(* Logix 5000 project; controller WWTP_SOLIDS_CLX vendor 1 type 14 code 54 rev 17.2; software revision 17.00; part 13 of 16 *)
(* tags used below, declared in another part *)
   Inp_ActuatorFault : BOOL;   // Valve Actuator Fault (overload, etc.), 0=OK, 1=Fault)
   Inp_OpenPermOK : BOOL;   // 1=Open Permissives OK, Valve can motor open
   Inp_OpenNBPermOK : BOOL;   // 1=Non-Bypassable Open Permissives OK, valve can motor open
   Inp_ClosePermOK : BOOL;   // 1=Close Permissives OK, Valve can motor closed
   Inp_CloseNBPermOK : BOOL;   // 1=Non-Bypassable Close Permissives OK, valve can motor closed
   Inp_IOFault : BOOL;   // Input Communication Status 0=OK, 1=fail
   Inp_Sim : BOOL;   // 1=Simulate working valve; 0=Open/Close/ Monitor actual valve
   Cfg_UseOpenLS : BOOL;   // 1=Valve Open LS should be used for failure checking
   Cfg_UseClosedLS : BOOL;   // 1=Valve Closed LS should be used for failure checking
   Cfg_HasStop : BOOL;   // 1=Stop output can be used to break local seal-in and stop valve motion
   Cfg_PCmdClear : BOOL;   // 1=Clear Program Commands on receipt 0=Leave Set
   Cfg_HasFullStallAlm : BOOL;   // 1=Full Stall Alarm exists and will be checked
   Cfg_HasTransitStallAlm : BOOL;   // 1=Transit Stall Alarm exists and will be checked
   Cfg_HasActuatorFaultAlm : BOOL;   // 1=Actuator Fault Alarm exists and will be checked
   Cfg_HasIOFaultAlm : BOOL;   // 1=I/O Fault Alarm exists and will be checked
   Cfg_FullStallResetReqd : BOOL;   // 1=Reset requied to clear Full Stall Alarm
   Cfg_TransitStallResetReqd : BOOL;   // 1=Reset required to clear Transit Stall Alarm
   Cfg_ActuatorFaultResetReqd : BOOL;   // 1=Reset required to clear Actuator Fault Alarm
   Cfg_IOFaultResetReqd : BOOL;   // 1=Reset required to clear I/O Fault Alarm
   Cfg_FullStallAckReqd : BOOL;   // 1=Acknowledge required for Full Stall Alarm
   Cfg_TransitStallAckReqd : BOOL;   // 1=Acknowledge required for Transit Stall Alarm
   Cfg_ActuatorFaultAckReqd : BOOL;   // 1=Acknowledge required for Actuator Fault Alarm
   Cfg_IOFaultAckReqd : BOOL;   // 1=Acknowledge required for I/O Fault Alarm
   Cfg_FullStallSeverity : SINT;   // Full Stall Alarm Severity 1=info 2=warn 3=excep 4=fault
   Cfg_TransitStallSeverity : SINT;   // Transit Stall Alarm Severity 1=info 2=warn 3=excep 4=fault
   Cfg_ActuatorFaultSeverity : SINT;   // Actuator Fault Alarm Severity 1=info 2=warn 3=excep 4=fault
   Cfg_IOFaultSeverity : SINT;   // I/O Fault Alarm Severity 1=info 2=warn 3=excep 4=fault
   PCmd_FullStallAck : BOOL;   // Program Command to Acknowledge Full Stall Alarm
   PCmd_FullStallInhibit : BOOL;   // Program Command to Inhibit Full Stall Alarm
   PCmd_FullStallUninhibit : BOOL;   // Program Command to Uninhibit Full Stall Alarm
   PCmd_TransitStallAck : BOOL;   // Program Command to Acknowledge Transit Stall Alarm
   PCmd_TransitStallInhibit : BOOL;   // Program Command to Inhibit Transit Stall Alarm
   PCmd_TransitStallUninhibit : BOOL;   // Program Command to Uninhibit Transit Stall Alarm
   PCmd_ActuatorFaultAck : BOOL;   // Program Command to Acknowledge Actuator Fault Alarm
   PCmd_ActuatorFaultInhibit : BOOL;   // Program Command to Inhibit Actuator Fault Alarm
   PCmd_ActuatorFaultUninhibit : BOOL;   // Program Command to Uninhibit Actuator Fault Alarm
   PCmd_IOFaultAck : BOOL;   // Program Command to Acknowledge I/O Fault Alarm
   PCmd_IOFaultInhibit : BOOL;   // Program Command to Inhibit I/O Fault Alarm
   PCmd_IOFaultUninhibit : BOOL;   // Program Command to Uninhibit I/O Fault Alarm
   Out_Open : BOOL;   // 1=Run actuator motor to OPEN Valve
   Out_Close : BOOL;   // 1=Run actuator motor to CLOSE Valve
   Out_Stop : BOOL;   // 1=Break seal-in circuit in actuator to STOP Valve motion
   Val_Notify : SINT;   // Current Alarm Level and Acknowledgement (enumeration)
   Sts_Closed : BOOL;   // 1=Valve requested to Close and is confirmed Closed
   Sts_CmdToOpen : BOOL;   // 1=Valve commanded to Open, has not yet moved off Open LS
   Sts_Opening : BOOL;   // 1=Valve requested to open and awaiting open feedback
   Sts_Opened : BOOL;   // 1=Valve requested to open and is confirmed Opened
   Sts_CmdToClose : BOOL;   // 1=Valve commanded to Close, has not yet moved off Closed LS
   Sts_Closing : BOOL;   // 1=Valve requested to Close and awaiting Closed feedback
   Sts_Stopped : BOOL;   // 1=Valve requested to Stop and is not at either end of travel
   Sts_Available : BOOL;   // 1=Valve available for control by automation (Prog)
   Sts_Bypass : BOOL;   // 1=Bypassable Interlocks and Permissives are Bypassed
   Sts_Disabled : BOOL;   // 1=Valve is Disabled
   Sts_LSFail : BOOL;   // 1=Limit Switch Overlap Failure
   Sts_Err : BOOL;   // 1=Error in Config: see detail bits for reason
   Err_Timer : BOOL;   // 1=Error in Config: Invalid Check or Pulse Time (use 0 to 2147483)
   Err_Sim : BOOL;   // 1=Error in Config: Simulation timer preset (use 0 to 2147483)
   Err_Alarm : BOOL;   // 1=Error in Config: Invalid Alarm Severity
   Sts_Hand : BOOL;   // 1=Mode is Hand (supersedes Maint, Ovrd, Prog, Oper)
   Sts_Maint : BOOL;   // 1=Mode is Maintenance (supersedes Ovrd, Prog, Oper)
   Sts_Ovrd : BOOL;   // 1=Mode is Override (supersedes Prog, Oper)
   Sts_Prog : BOOL;   // 1=Mode is Program (auto)
   Sts_Oper : BOOL;   // 1=Mode is Operator (manual)
   Sts_ProgOperLock : BOOL;   // 1=Program or Operator has requested Mode Lock
   Sts_FullStall : BOOL;   // 1=Valve Full Stall (failed to move at all) (One-Shot)
   Alm_FullStall : BOOL;   // 1=Valve Full Stall (failed to move at all) Alarm
   Ack_FullStall : BOOL;   // 1=Full Stall Alarm has been acknowledged
   Sts_FullStallDisabled : BOOL;   // 1=Full Stall Alarm has been disabled (will not be sent)
   Sts_FullStallInhibited : BOOL;   // 1=Full Stall Alarm has been inhibited by logic
   Sts_FullStallSuppressed : BOOL;   // 1=Full Stall Alarm has been suppressed (logged only)
   Sts_TransitStall : BOOL;   // 1=Valve Transit Stall (did not reach target position) (One-Shot)
   Alm_TransitStall : BOOL;   // 1=Valve Transit Stall (did not reach target pos.) Alarm
   Ack_TransitStall : BOOL;   // 1=Transit Stall Alarm has been acknowledged
   Sts_TransitStallDisabled : BOOL;   // 1=Transit Stall Alarm has been disabled (will not be sent)
   Sts_TransitStallInhibited : BOOL;   // 1=Transit Stall Alarm has been inhibited by logic
   Sts_TransitStallSuppressed : BOOL;   // 1=Transit Stall Alarm has been suppressed (logged only)
   Sts_ActuatorFault : BOOL;   // 1=Actuator Fault detected (input)
   Alm_ActuatorFault : BOOL;   // 1=Alarm: Actuator Fault Detected
   Ack_ActuatorFault : BOOL;   // 1=Actuator Fault Alarm has been acknowledged
   Sts_ActuatorFaultDisabled : BOOL;   // 1=Actuator Fault Alarm is Disabled (not saved or sent)
   Sts_ActuatorFaultInhibited : BOOL;   // 1=Actuator Fault Alarm has been inhibited by logic
   Sts_ActuatorFaultSuppressed : BOOL;   // 1=Actuator Fault Alarm has been suppressed (logged only)
   Sts_IOFault : BOOL;   // I/O Comm Fault Status (0=OK, 1=Bad)
   Alm_IOFault : BOOL;   // 1=I/O Fault Alarm
   Ack_IOFault : BOOL;   // 1=I/O Fault Alarm has been acknowledged
   Sts_IOFaultDisabled : BOOL;   // 1=I/O Fault Alarm is Disabled (not saved or sent)
   Sts_IOFaultInhibited : BOOL;   // 1=I/O Fault Alarm has been inhibited by logic
   Sts_IOFaultSuppressed : BOOL;   // 1=I/O Fault Alarm has been suppressed (logged only)
   Rdy_Open : BOOL;   // 1=Ready to receive OCmd_Open (enables HMI button)
   Rdy_Close : BOOL;   // 1=Ready to receive OCmd_Close (enables HMI button)
   Rdy_Stop : BOOL;   // 1=Ready to receive OCmd_Stop (enables HMI button)
   Rdy_Bypass : BOOL;   // 1=Ready to receive OCmd_Bypass (enables HMI button)
   Rdy_Check : BOOL;   // 1=Ready to receive OCmd_Check (enables HMI button)
   Rdy_Disable : BOOL;   // 1=Ready to receive MCmd_Disable (enables HMI button)
   Rdy_Enable : BOOL;   // 1=Ready to receive MCmd_Enable (enables HMI button)
   Rdy_Reset : BOOL;   // 1=Ready to receive OCmd_Reset (enables HMI button)
   Mode : P_Mode;   // Valve Mode Selection
   IOFault : P_Alarm;   // I/O Fault Alarm
   ActuatorFault : P_Alarm;   // Actuator Fault Alarm
   TransitStall : P_Alarm;   // Valve Transit Stall (moved but did not reach target) Alarm
   FullStall : P_Alarm;   // Valve Full Stall (did not move) Alarm
   Wrk_Open : BOOL;   // 1=Requested to OPEN Valve
   Wrk_Fault : BOOL;   // 1=a Valve Fault has been detected
   Wrk_OpenFdbk : BOOL;   // 1=LS Feedback shows valve confirmed open
   Wrk_Notify : DINT;   // Buffer for building Val_Notify
   Wrk_Bypass : BOOL;   // Internal Bypassable Permissives and Interlocks are Bypassed flag
   Wrk_Disabled : BOOL;   // Internal Valve is Disabled
   Wrk_ClosedFdbk : BOOL;   // 1=LS Feedback shows valve confirmed closed
   Wrk_LSFailFdbk : BOOL;   // 1=LS Feedback shows Limit Switch Failure
   Wrk_TravelFdbk : BOOL;   // 1=LS Feedback shows Valve is Traveling
   Wrk_Stop : BOOL;   // 1=Requested to STOP Valve
   Wrk_Close : BOOL;   // 1-Requested to CLOSE Valve
   Wrk_StopPulseT : TIMER;   // Timer for Out_Stop pulse time
   Wrk_ClosePulseT : TIMER;   // Timer for Out_Close pulse time
   Wrk_OpenPulseT : TIMER;   // Timer for Out_Open pulse time
   Wrk_TransitStallT : TIMER;   // Timer for Transit Stall Check
(* P_ValveMO, continued *)

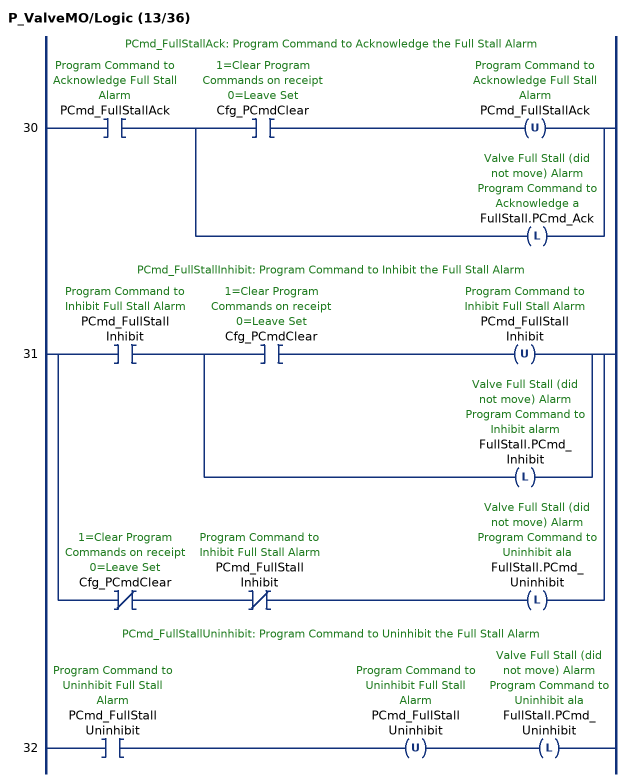
   [picture p269: P_ValveMO/Logic rungs 30-32]
   // PCmd_FullStallAck: Program Command to Acknowledge the Full Stall Alarm
   30: XIC(PCmd_FullStallAck)[XIC(Cfg_PCmdClear) OTU(PCmd_FullStallAck) ,OTL(FullStall.PCmd_Ack) ];
   // PCmd_FullStallInhibit: Program Command to Inhibit the Full Stall Alarm
   31: [XIC(PCmd_FullStallInhibit) [XIC(Cfg_PCmdClear) OTU(PCmd_FullStallInhibit) ,OTL(FullStall.PCmd_Inhibit) ] ,XIO(Cfg_PCmdClear) XIO(PCmd_FullStallInhibit) OTL(FullStall.PCmd_Uninhibit) ];
   // PCmd_FullStallUninhibit: Program Command to Uninhibit the Full Stall Alarm
   32: XIC(PCmd_FullStallUninhibit)OTU(PCmd_FullStallUninhibit)OTL(FullStall.PCmd_Uninhibit);
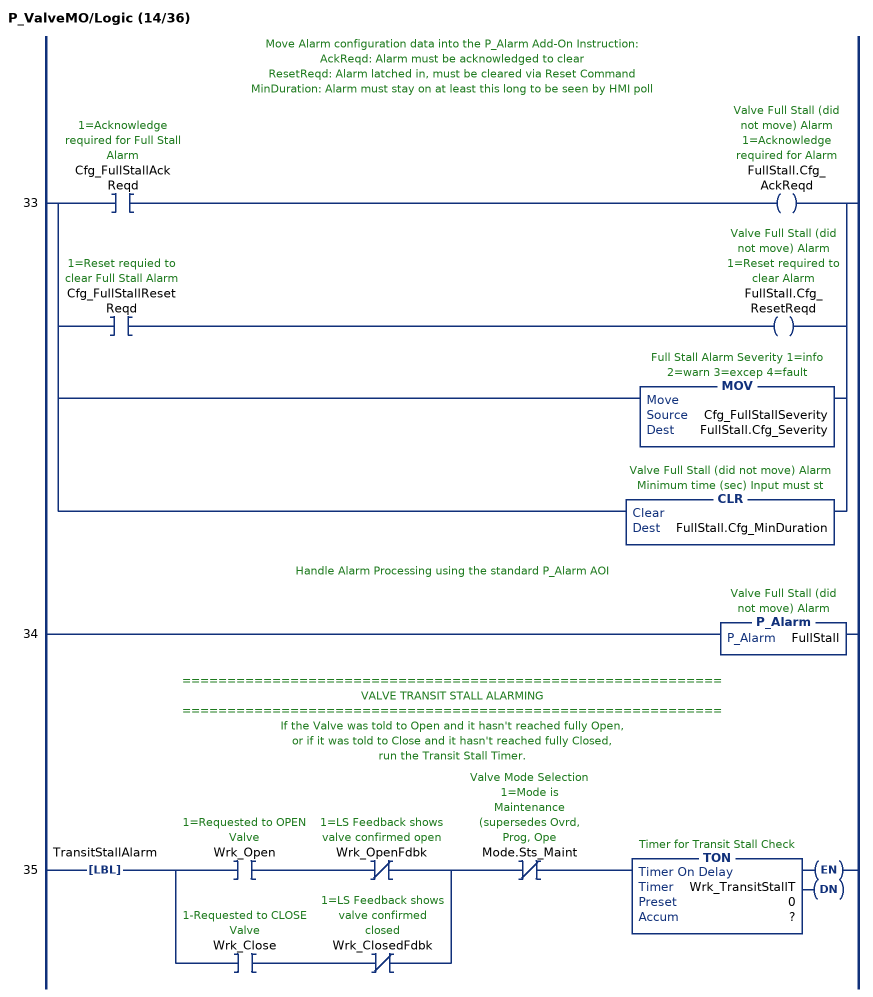
   // Move Alarm configuration data into the P_Alarm Add-On Instruction:
   // AckReqd: Alarm must be acknowledged to clear
   // ResetReqd: Alarm latched in, must be cleared via Reset Command
   // MinDuration: Alarm must stay on at least this long to be seen by HMI poll
   33: [XIC(Cfg_FullStallAckReqd) OTE(FullStall.Cfg_AckReqd) ,XIC(Cfg_FullStallResetReqd) OTE(FullStall.Cfg_ResetReqd) ,MOV(Cfg_FullStallSeverity,FullStall.Cfg_Severity) ,CLR(FullStall.Cfg_MinDuration) ];
   // Handle Alarm Processing using the standard P_Alarm AOI
   34: P_Alarm(FullStall);
   // ============================================================
   // VALVE TRANSIT STALL ALARMING
   // ============================================================
   // If the Valve was told to Open and it hasn't reached fully Open,
   // or if it was told to Close and it hasn't reached fully Closed,
   // run the Transit Stall Timer.
   35: LBL(TransitStallAlarm)[XIC(Wrk_Open) XIO(Wrk_OpenFdbk) ,XIC(Wrk_Close) XIO(Wrk_ClosedFdbk) ]XIO(Mode.Sts_Maint)TON(Wrk_TransitStallT,?,?);
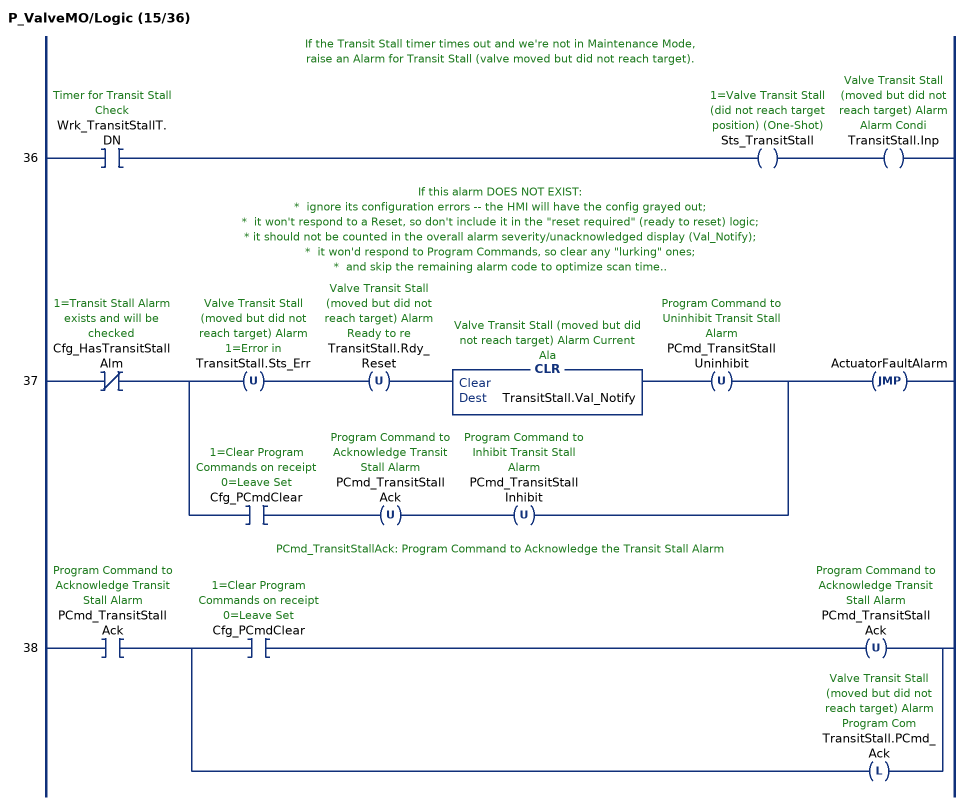
   // If the Transit Stall timer times out and we're not in Maintenance Mode,
   // raise an Alarm for Transit Stall (valve moved but did not reach target).
   36: XIC(Wrk_TransitStallT.DN)OTE(Sts_TransitStall)OTE(TransitStall.Inp);
   // If this alarm DOES NOT EXIST:
   // *  ignore its configuration errors -- the HMI will have the config grayed out;
   // *  it won't respond to a Reset, so don't include it in the "reset required" (ready to reset) logic;
   // * it should not be counted in the overall alarm severity/unacknowledged display (Val_Notify);
   // *  it won'd respond to Program Commands, so clear any "lurking" ones;
   // *  and skip the remaining alarm code to optimize scan time..
   37: XIO(Cfg_HasTransitStallAlm)[OTU(TransitStall.Sts_Err) OTU(TransitStall.Rdy_Reset) CLR(TransitStall.Val_Notify) OTU(PCmd_TransitStallUninhibit) ,XIC(Cfg_PCmdClear) OTU(PCmd_TransitStallAck) OTU(PCmd_TransitStallInhibit) ]JMP(ActuatorFaultAlarm);
   // PCmd_TransitStallAck: Program Command to Acknowledge the Transit Stall Alarm
   38: XIC(PCmd_TransitStallAck)[XIC(Cfg_PCmdClear) OTU(PCmd_TransitStallAck) ,OTL(TransitStall.PCmd_Ack) ];
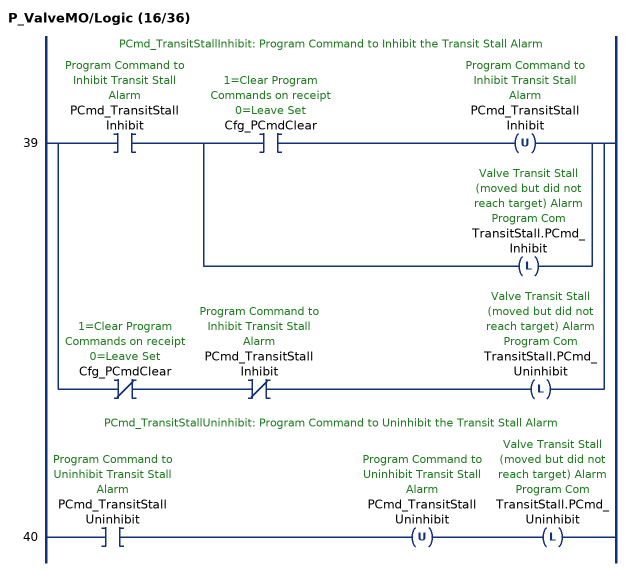
   // PCmd_TransitStallInhibit: Program Command to Inhibit the Transit Stall Alarm
   39: [XIC(PCmd_TransitStallInhibit) [XIC(Cfg_PCmdClear) OTU(PCmd_TransitStallInhibit) ,OTL(TransitStall.PCmd_Inhibit) ] ,XIO(Cfg_PCmdClear) XIO(PCmd_TransitStallInhibit) OTL(TransitStall.PCmd_Uninhibit) ];
   // PCmd_TransitStallUninhibit: Program Command to Uninhibit the Transit Stall Alarm
   40: XIC(PCmd_TransitStallUninhibit)OTU(PCmd_TransitStallUninhibit)OTL(TransitStall.PCmd_Uninhibit);
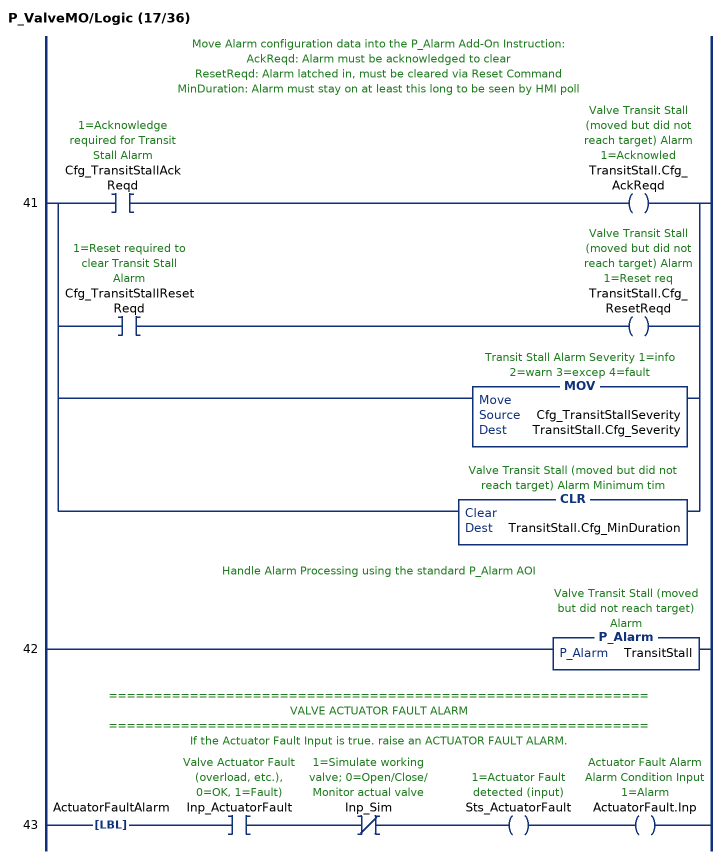
   // Move Alarm configuration data into the P_Alarm Add-On Instruction:
   // AckReqd: Alarm must be acknowledged to clear
   // ResetReqd: Alarm latched in, must be cleared via Reset Command
   // MinDuration: Alarm must stay on at least this long to be seen by HMI poll
   41: [XIC(Cfg_TransitStallAckReqd) OTE(TransitStall.Cfg_AckReqd) ,XIC(Cfg_TransitStallResetReqd) OTE(TransitStall.Cfg_ResetReqd) ,MOV(Cfg_TransitStallSeverity,TransitStall.Cfg_Severity) ,CLR(TransitStall.Cfg_MinDuration) ];
   // Handle Alarm Processing using the standard P_Alarm AOI
   42: P_Alarm(TransitStall);
   // ============================================================
   // VALVE ACTUATOR FAULT ALARM
   // ============================================================
   // If the Actuator Fault Input is true. raise an ACTUATOR FAULT ALARM.
   43: LBL(ActuatorFaultAlarm)XIC(Inp_ActuatorFault)XIO(Inp_Sim)OTE(Sts_ActuatorFault)OTE(ActuatorFault.Inp);
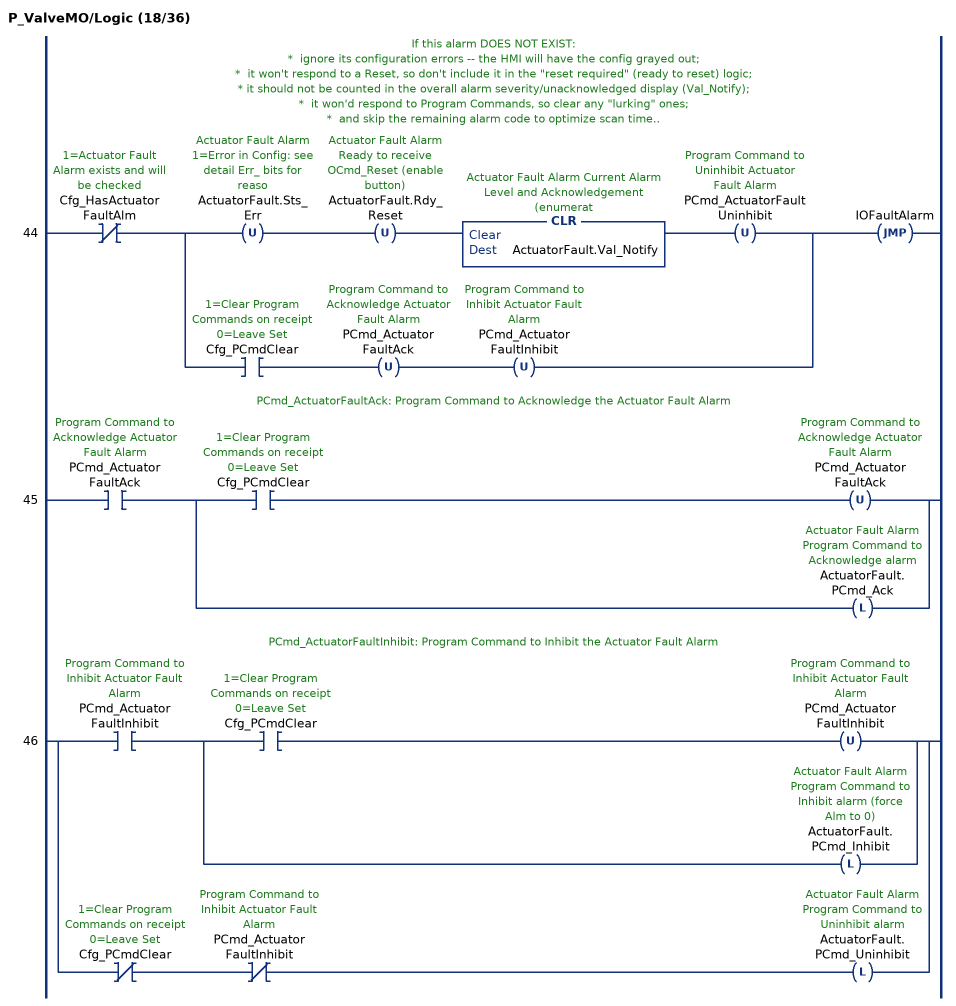
   // If this alarm DOES NOT EXIST:
   // *  ignore its configuration errors -- the HMI will have the config grayed out;
   // *  it won't respond to a Reset, so don't include it in the "reset required" (ready to reset) logic;
   // * it should not be counted in the overall alarm severity/unacknowledged display (Val_Notify);
   // *  it won'd respond to Program Commands, so clear any "lurking" ones;
   // *  and skip the remaining alarm code to optimize scan time..
   44: XIO(Cfg_HasActuatorFaultAlm)[OTU(ActuatorFault.Sts_Err) OTU(ActuatorFault.Rdy_Reset) CLR(ActuatorFault.Val_Notify) OTU(PCmd_ActuatorFaultUninhibit) ,XIC(Cfg_PCmdClear) OTU(PCmd_ActuatorFaultAck) OTU(PCmd_ActuatorFaultInhibit) ]JMP(IOFaultAlarm);
   // PCmd_ActuatorFaultAck: Program Command to Acknowledge the Actuator Fault Alarm
   45: XIC(PCmd_ActuatorFaultAck)[XIC(Cfg_PCmdClear) OTU(PCmd_ActuatorFaultAck) ,OTL(ActuatorFault.PCmd_Ack) ];
   // PCmd_ActuatorFaultInhibit: Program Command to Inhibit the Actuator Fault Alarm
   46: [XIC(PCmd_ActuatorFaultInhibit) [XIC(Cfg_PCmdClear) OTU(PCmd_ActuatorFaultInhibit) ,OTL(ActuatorFault.PCmd_Inhibit) ] ,XIO(Cfg_PCmdClear) XIO(PCmd_ActuatorFaultInhibit) OTL(ActuatorFault.PCmd_Uninhibit) ];
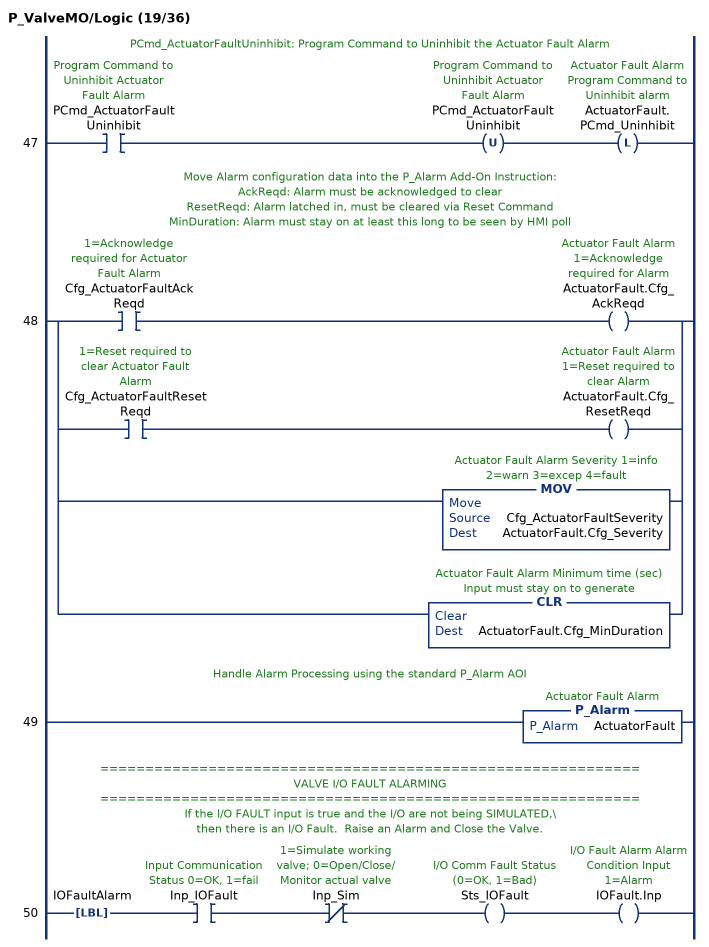
   // PCmd_ActuatorFaultUninhibit: Program Command to Uninhibit the Actuator Fault Alarm
   47: XIC(PCmd_ActuatorFaultUninhibit)OTU(PCmd_ActuatorFaultUninhibit)OTL(ActuatorFault.PCmd_Uninhibit);
   // Move Alarm configuration data into the P_Alarm Add-On Instruction:
   // AckReqd: Alarm must be acknowledged to clear
   // ResetReqd: Alarm latched in, must be cleared via Reset Command
   // MinDuration: Alarm must stay on at least this long to be seen by HMI poll
   48: [XIC(Cfg_ActuatorFaultAckReqd) OTE(ActuatorFault.Cfg_AckReqd) ,XIC(Cfg_ActuatorFaultResetReqd) OTE(ActuatorFault.Cfg_ResetReqd) ,MOV(Cfg_ActuatorFaultSeverity,ActuatorFault.Cfg_Severity) ,CLR(ActuatorFault.Cfg_MinDuration) ];
   // Handle Alarm Processing using the standard P_Alarm AOI
   49: P_Alarm(ActuatorFault);
   // ============================================================
   // VALVE I/O FAULT ALARMING
   // ============================================================
   // If the I/O FAULT input is true and the I/O are not being SIMULATED,\
   // then there is an I/O Fault.  Raise an Alarm and Close the Valve.
   50: LBL(IOFaultAlarm)XIC(Inp_IOFault)XIO(Inp_Sim)OTE(Sts_IOFault)OTE(IOFault.Inp);
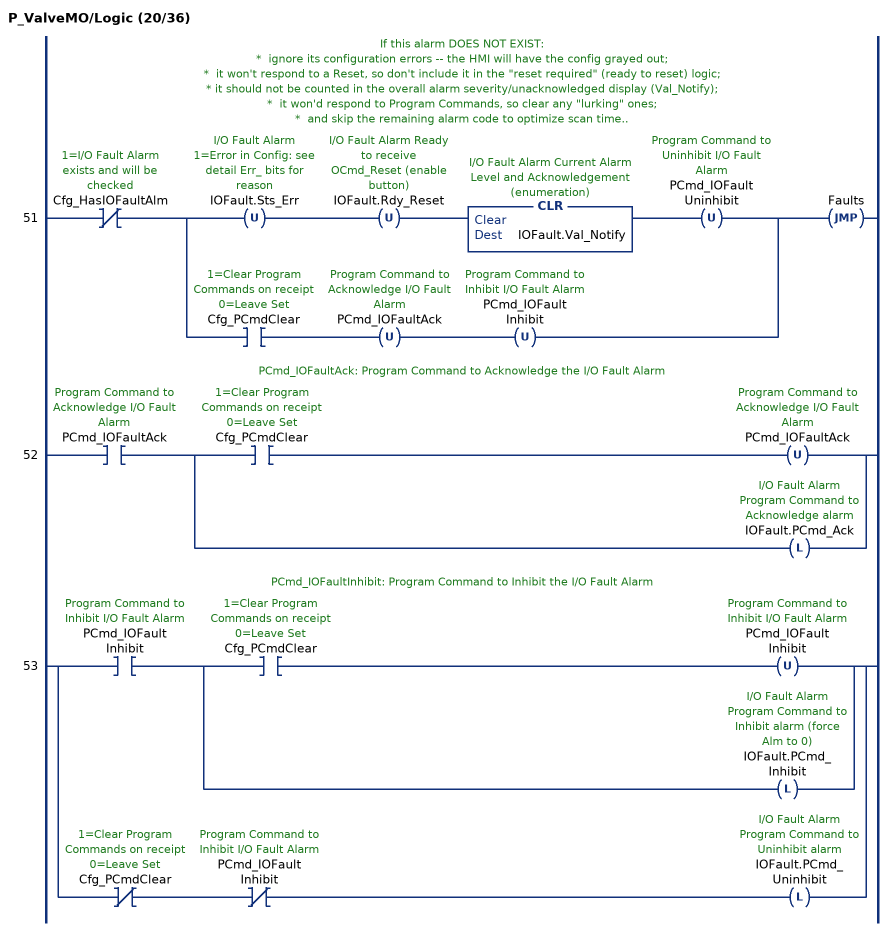
   // If this alarm DOES NOT EXIST:
   // *  ignore its configuration errors -- the HMI will have the config grayed out;
   // *  it won't respond to a Reset, so don't include it in the "reset required" (ready to reset) logic;
   // * it should not be counted in the overall alarm severity/unacknowledged display (Val_Notify);
   // *  it won'd respond to Program Commands, so clear any "lurking" ones;
   // *  and skip the remaining alarm code to optimize scan time..
   51: XIO(Cfg_HasIOFaultAlm)[OTU(IOFault.Sts_Err) OTU(IOFault.Rdy_Reset) CLR(IOFault.Val_Notify) OTU(PCmd_IOFaultUninhibit) ,XIC(Cfg_PCmdClear) OTU(PCmd_IOFaultAck) OTU(PCmd_IOFaultInhibit) ]JMP(Faults);
   // PCmd_IOFaultAck: Program Command to Acknowledge the I/O Fault Alarm
   52: XIC(PCmd_IOFaultAck)[XIC(Cfg_PCmdClear) OTU(PCmd_IOFaultAck) ,OTL(IOFault.PCmd_Ack) ];
   // PCmd_IOFaultInhibit: Program Command to Inhibit the I/O Fault Alarm
   53: [XIC(PCmd_IOFaultInhibit) [XIC(Cfg_PCmdClear) OTU(PCmd_IOFaultInhibit) ,OTL(IOFault.PCmd_Inhibit) ] ,XIO(Cfg_PCmdClear) XIO(PCmd_IOFaultInhibit) OTL(IOFault.PCmd_Uninhibit) ];
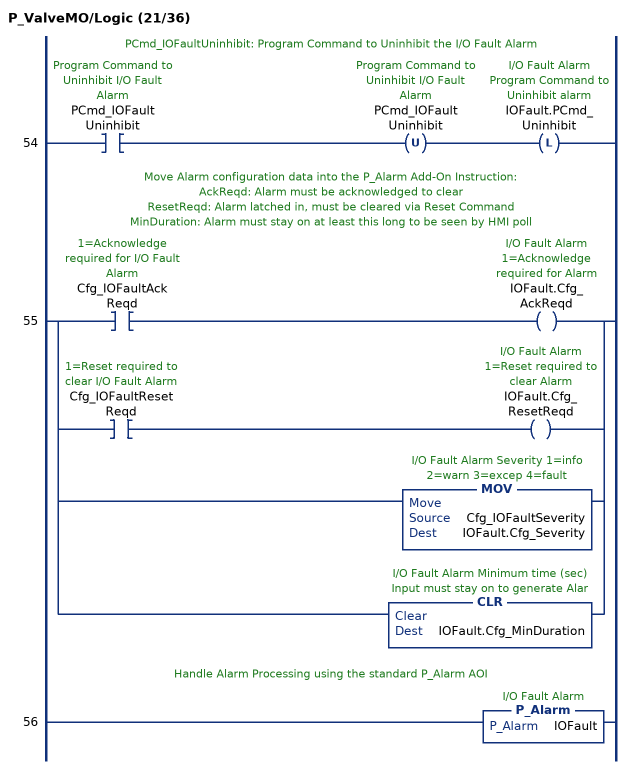
   // PCmd_IOFaultUninhibit: Program Command to Uninhibit the I/O Fault Alarm
   54: XIC(PCmd_IOFaultUninhibit)OTU(PCmd_IOFaultUninhibit)OTL(IOFault.PCmd_Uninhibit);
   // Move Alarm configuration data into the P_Alarm Add-On Instruction:
   // AckReqd: Alarm must be acknowledged to clear
   // ResetReqd: Alarm latched in, must be cleared via Reset Command
   // MinDuration: Alarm must stay on at least this long to be seen by HMI poll
   55: [XIC(Cfg_IOFaultAckReqd) OTE(IOFault.Cfg_AckReqd) ,XIC(Cfg_IOFaultResetReqd) OTE(IOFault.Cfg_ResetReqd) ,MOV(Cfg_IOFaultSeverity,IOFault.Cfg_Severity) ,CLR(IOFault.Cfg_MinDuration) ];
   // Handle Alarm Processing using the standard P_Alarm AOI
   56: P_Alarm(IOFault);
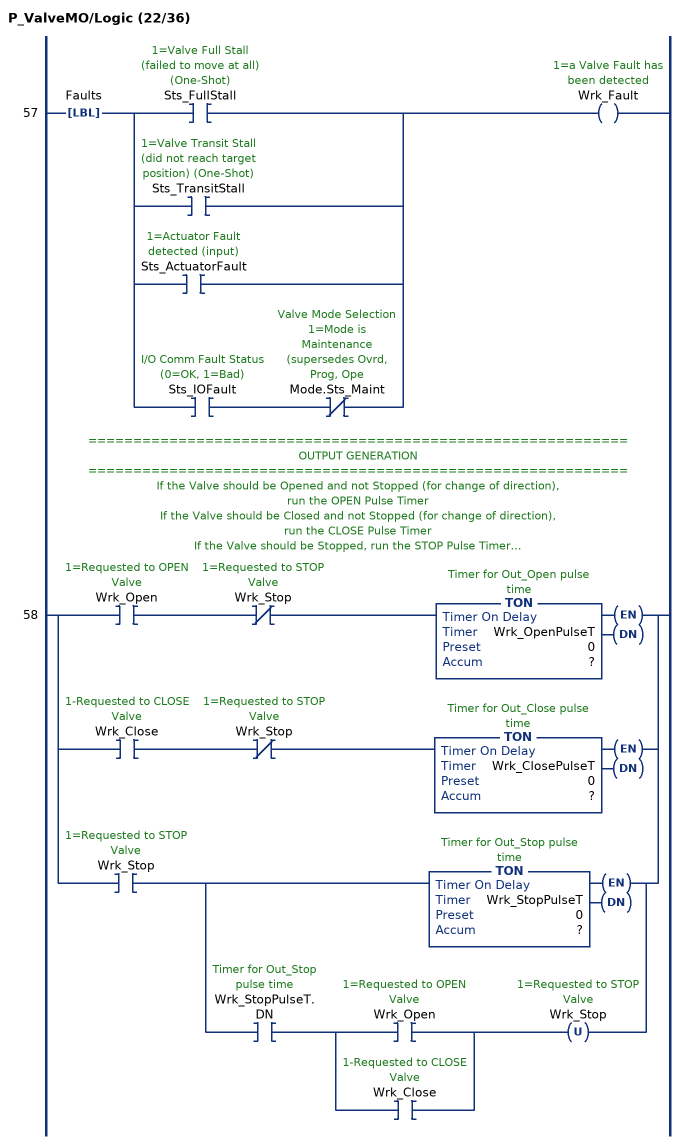
   57: LBL(Faults)[XIC(Sts_FullStall) ,XIC(Sts_TransitStall) ,XIC(Sts_ActuatorFault) ,XIC(Sts_IOFault) XIO(Mode.Sts_Maint) ]OTE(Wrk_Fault);
   // ============================================================
   // OUTPUT GENERATION
   // ============================================================
   // If the Valve should be Opened and not Stopped (for change of direction),
   // run the OPEN Pulse Timer
   // If the Valve should be Closed and not Stopped (for change of direction),
   // run the CLOSE Pulse Timer
   // If the Valve should be Stopped, run the STOP Pulse Timer.
   // When the timer is DONE, if we ARE doing a Change of Direction,
   // continue by Opening or Closing the valve (as appropriate) and turn off the STOP request.
   58: [XIC(Wrk_Open) XIO(Wrk_Stop) TON(Wrk_OpenPulseT,?,?) ,XIC(Wrk_Close) XIO(Wrk_Stop) TON(Wrk_ClosePulseT,?,?) ,XIC(Wrk_Stop) [TON(Wrk_StopPulseT,?,?) ,XIC(Wrk_StopPulseT.DN) [XIC(Wrk_Open) ,XIC(Wrk_Close) ] OTU(Wrk_Stop) ] ];
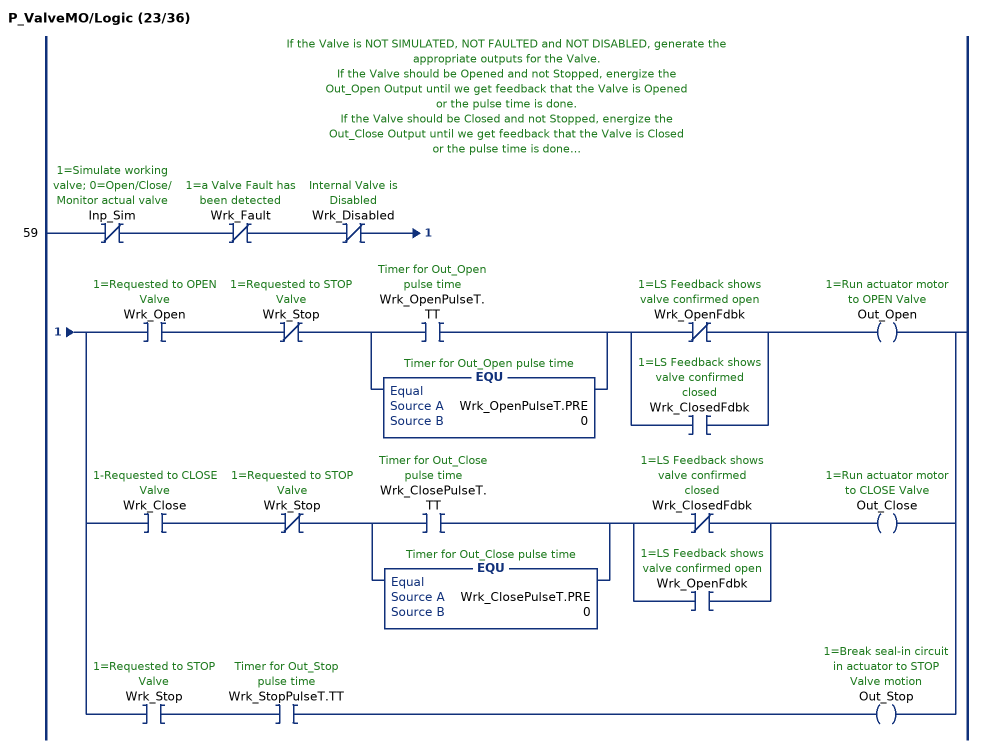
   // If the Valve is NOT SIMULATED, NOT FAULTED and NOT DISABLED, generate the
   // appropriate outputs for the Valve.
   // If the Valve should be Opened and not Stopped, energize the
   // Out_Open Output until we get feedback that the Valve is Opened
   // or the pulse time is done.
   // If the Valve should be Closed and not Stopped, energize the
   // Out_Close Output until we get feedback that the Valve is Closed
   // or the pulse time is done.
   // If the Valve should be Stopped, energize Out_Stop for the full pulse duration.
   59: XIO(Inp_Sim)XIO(Wrk_Fault)XIO(Wrk_Disabled)[XIC(Wrk_Open) XIO(Wrk_Stop) [XIC(Wrk_OpenPulseT.TT) ,EQU(Wrk_OpenPulseT.PRE,0) ] [XIO(Wrk_OpenFdbk) ,XIC(Wrk_ClosedFdbk) ] OTE(Out_Open) ,XIC(Wrk_Close) XIO(Wrk_Stop) [XIC(Wrk_ClosePulseT.TT) ,EQU(Wrk_ClosePulseT.PRE,0) ] [XIO(Wrk_ClosedFdbk) ,XIC(Wrk_OpenFdbk) ] OTE(Out_Close) ,XIC(Wrk_Stop) XIC(Wrk_StopPulseT.TT) OTE(Out_Stop) ];
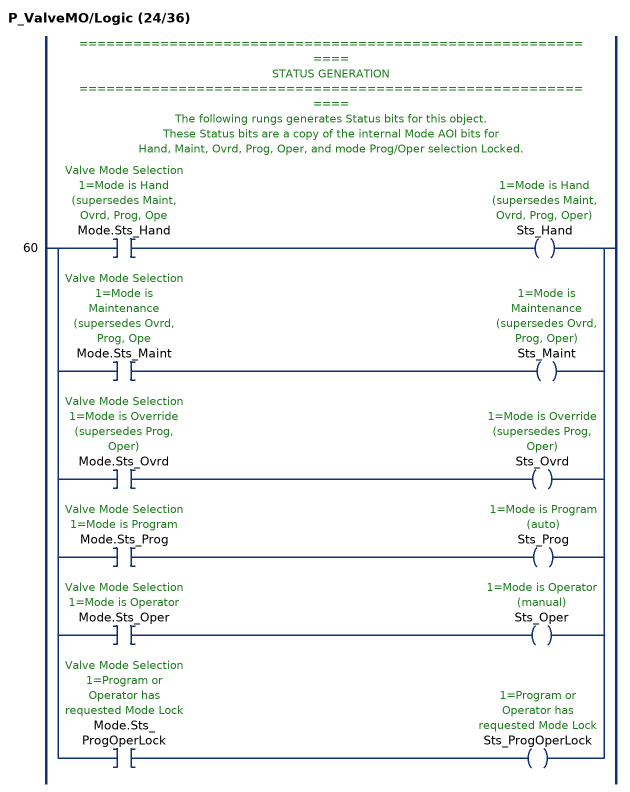
   // ============================================================
   // STATUS GENERATION
   // ============================================================
   // The following rungs generates Status bits for this object.
   // These Status bits are a copy of the internal Mode AOI bits for
   // Hand, Maint, Ovrd, Prog, Oper, and mode Prog/Oper selection Locked.
   60: [XIC(Mode.Sts_Hand) OTE(Sts_Hand) ,XIC(Mode.Sts_Maint) OTE(Sts_Maint) ,XIC(Mode.Sts_Ovrd) OTE(Sts_Ovrd) ,XIC(Mode.Sts_Prog) OTE(Sts_Prog) ,XIC(Mode.Sts_Oper) OTE(Sts_Oper) ,XIC(Mode.Sts_ProgOperLock) OTE(Sts_ProgOperLock) ];
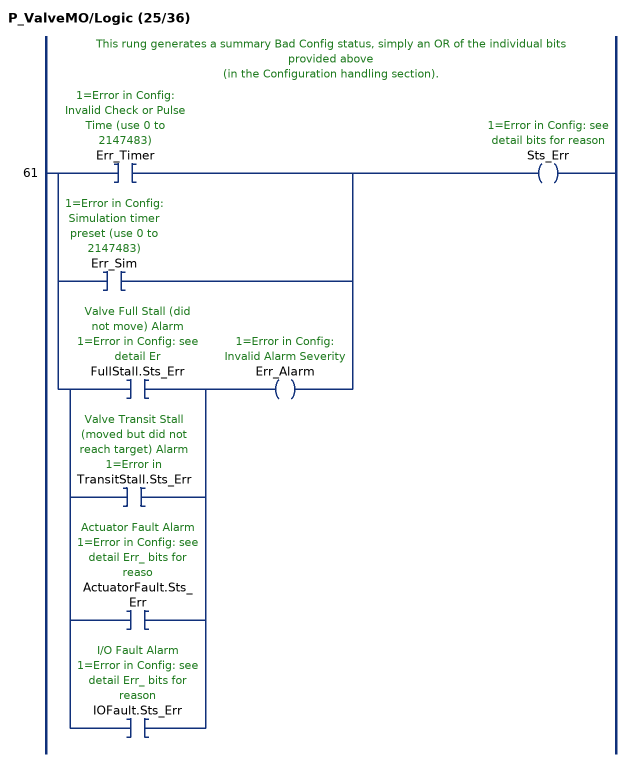
   // This rung generates a summary Bad Config status, simply an OR of the individual bits provided above
   // (in the Configuration handling section).
   61: [XIC(Err_Timer) ,XIC(Err_Sim) ,[XIC(FullStall.Sts_Err) ,XIC(TransitStall.Sts_Err) ,XIC(ActuatorFault.Sts_Err) ,XIC(IOFault.Sts_Err) ] OTE(Err_Alarm) ]OTE(Sts_Err);
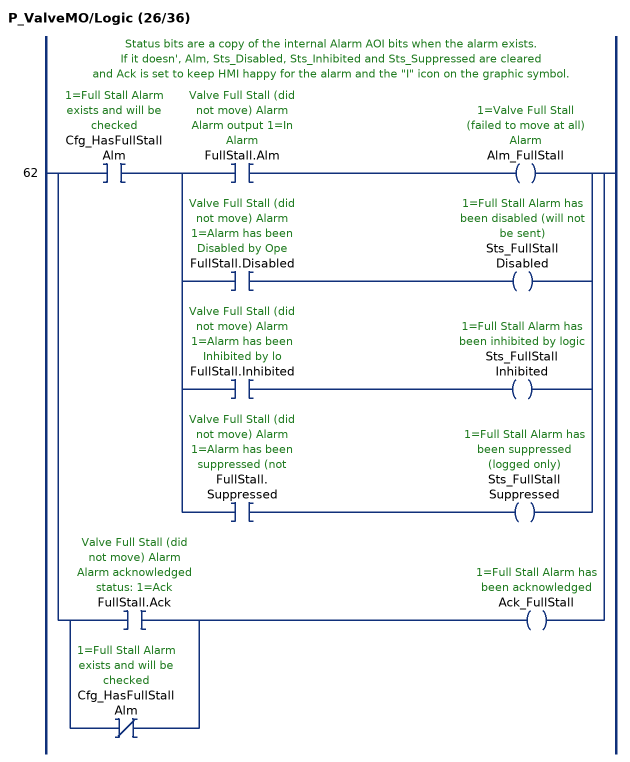
   // Status bits are a copy of the internal Alarm AOI bits when the alarm exists.
   // If it doesn', Alm, Sts_Disabled, Sts_Inhibited and Sts_Suppressed are cleared
   // and Ack is set to keep HMI happy for the alarm and the "I" icon on the graphic symbol.
   62: [XIC(Cfg_HasFullStallAlm) [XIC(FullStall.Alm) OTE(Alm_FullStall) ,XIC(FullStall.Disabled) OTE(Sts_FullStallDisabled) ,XIC(FullStall.Inhibited) OTE(Sts_FullStallInhibited) ,XIC(FullStall.Suppressed) OTE(Sts_FullStallSuppressed) ] ,[XIC(FullStall.Ack) ,XIO(Cfg_HasFullStallAlm) ] OTE(Ack_FullStall) ];
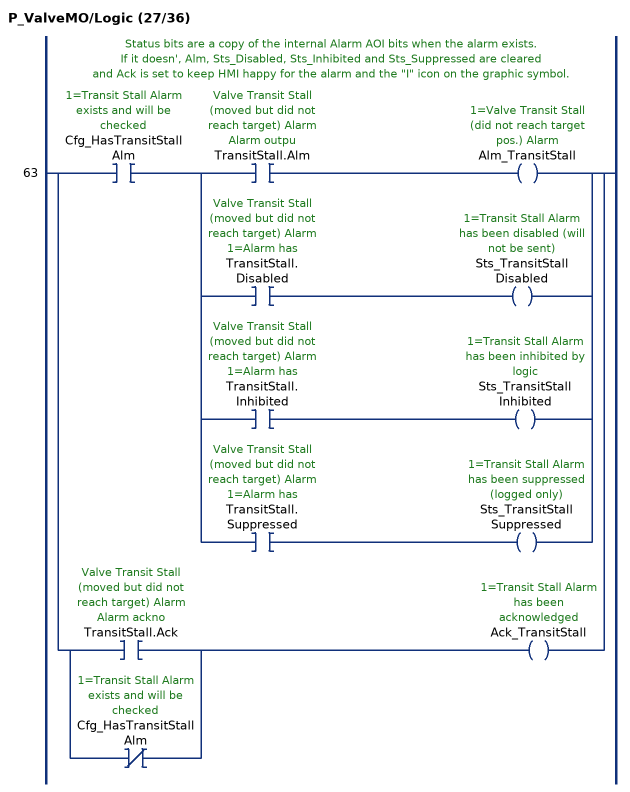
   // Status bits are a copy of the internal Alarm AOI bits when the alarm exists.
   // If it doesn', Alm, Sts_Disabled, Sts_Inhibited and Sts_Suppressed are cleared
   // and Ack is set to keep HMI happy for the alarm and the "I" icon on the graphic symbol.
   63: [XIC(Cfg_HasTransitStallAlm) [XIC(TransitStall.Alm) OTE(Alm_TransitStall) ,XIC(TransitStall.Disabled) OTE(Sts_TransitStallDisabled) ,XIC(TransitStall.Inhibited) OTE(Sts_TransitStallInhibited) ,XIC(TransitStall.Suppressed) OTE(Sts_TransitStallSuppressed) ] ,[XIC(TransitStall.Ack) ,XIO(Cfg_HasTransitStallAlm) ] OTE(Ack_TransitStall) ];
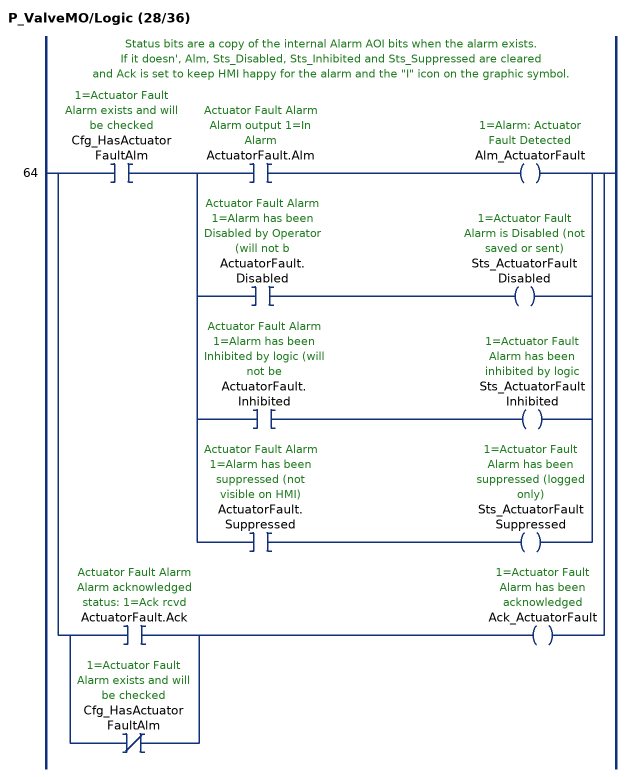
   // Status bits are a copy of the internal Alarm AOI bits when the alarm exists.
   // If it doesn', Alm, Sts_Disabled, Sts_Inhibited and Sts_Suppressed are cleared
   // and Ack is set to keep HMI happy for the alarm and the "I" icon on the graphic symbol.
   64: [XIC(Cfg_HasActuatorFaultAlm) [XIC(ActuatorFault.Alm) OTE(Alm_ActuatorFault) ,XIC(ActuatorFault.Disabled) OTE(Sts_ActuatorFaultDisabled) ,XIC(ActuatorFault.Inhibited) OTE(Sts_ActuatorFaultInhibited) ,XIC(ActuatorFault.Suppressed) OTE(Sts_ActuatorFaultSuppressed) ] ,[XIC(ActuatorFault.Ack) ,XIO(Cfg_HasActuatorFaultAlm) ] OTE(Ack_ActuatorFault) ];
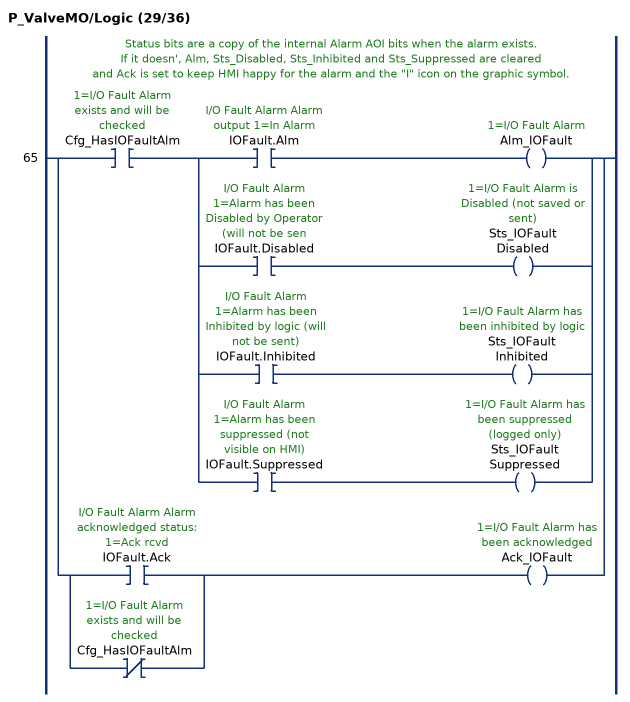
   // Status bits are a copy of the internal Alarm AOI bits when the alarm exists.
   // If it doesn', Alm, Sts_Disabled, Sts_Inhibited and Sts_Suppressed are cleared
   // and Ack is set to keep HMI happy for the alarm and the "I" icon on the graphic symbol.
   65: [XIC(Cfg_HasIOFaultAlm) [XIC(IOFault.Alm) OTE(Alm_IOFault) ,XIC(IOFault.Disabled) OTE(Sts_IOFaultDisabled) ,XIC(IOFault.Inhibited) OTE(Sts_IOFaultInhibited) ,XIC(IOFault.Suppressed) OTE(Sts_IOFaultSuppressed) ] ,[XIC(IOFault.Ack) ,XIO(Cfg_HasIOFaultAlm) ] OTE(Ack_IOFault) ];
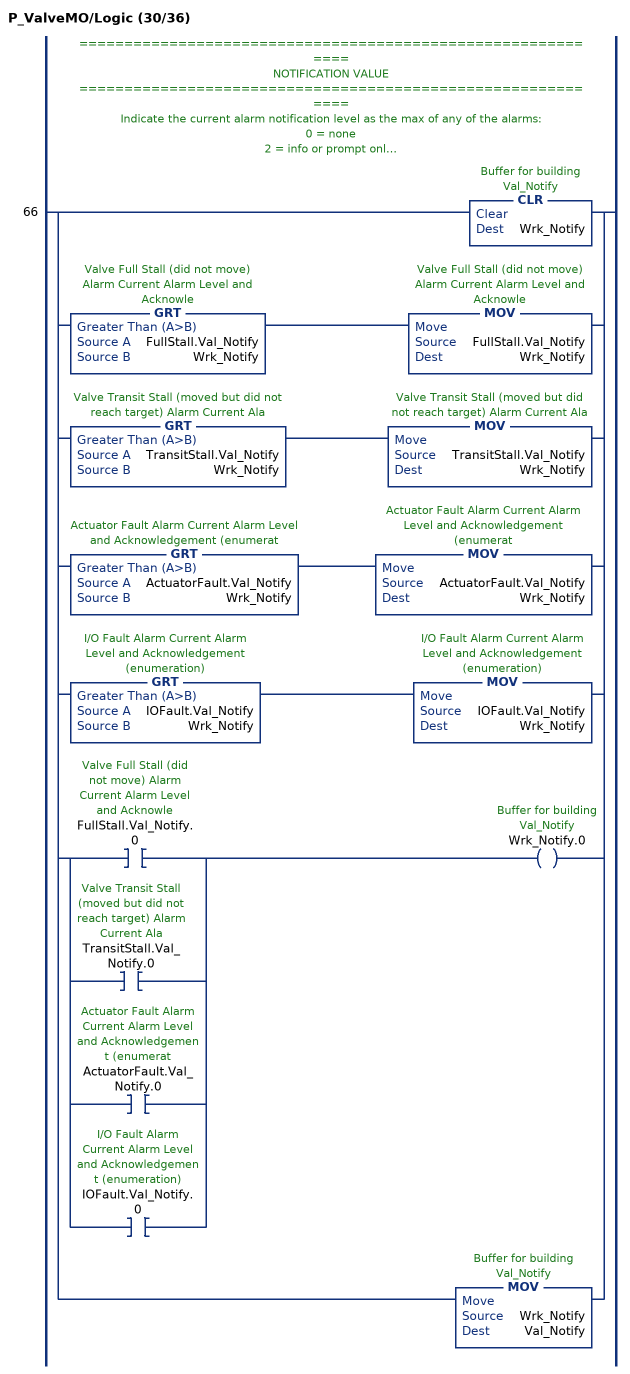
   // ============================================================
   // NOTIFICATION VALUE
   // ============================================================
   // Indicate the current alarm notification level as the max of any of the alarms:
   // 0 = none
   // 2 = info or prompt only
   // 4 = warning
   // 6 = exception (equipment impact)
   // 8 = fault (equipment failure)
   // Add one for any unsuppressed alarm that is not acknowledged (for blink).
   66: [CLR(Wrk_Notify) ,GRT(FullStall.Val_Notify,Wrk_Notify) MOV(FullStall.Val_Notify,Wrk_Notify) ,GRT(TransitStall.Val_Notify,Wrk_Notify) MOV(TransitStall.Val_Notify,Wrk_Notify) ,GRT(ActuatorFault.Val_Notify,Wrk_Notify) MOV(ActuatorFault.Val_Notify,Wrk_Notify) ,GRT(IOFault.Val_Notify,Wrk_Notify) MOV(IOFault.Val_Notify,Wrk_Notify) ,[XIC(FullStall.Val_Notify.0) ,XIC(TransitStall.Val_Notify.0) ,XIC(ActuatorFault.Val_Notify.0) ,XIC(IOFault.Val_Notify.0) ] OTE(Wrk_Notify.0) ,MOV(Wrk_Notify,Val_Notify) ];
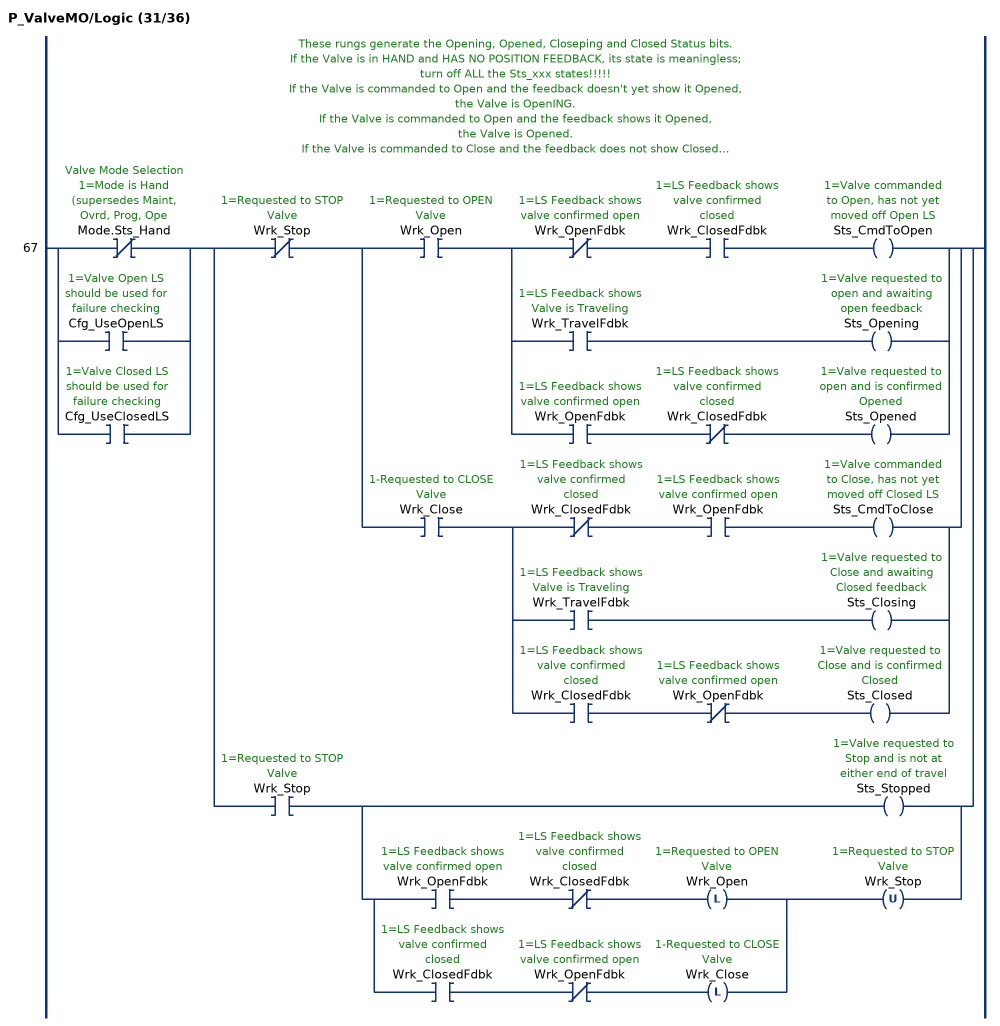
   // These rungs generate the Opening, Opened, Closeping and Closed Status bits.
   // If the Valve is in HAND and HAS NO POSITION FEEDBACK, its state is meaningless;
   // turn off ALL the Sts_xxx states!!!!!
   // If the Valve is commanded to Open and the feedback doesn't yet show it Opened,
   // the Valve is OpenING.
   // If the Valve is commanded to Open and the feedback shows it Opened,
   // the Valve is Opened.
   // If the Valve is commanded to Close and the feedback does not show Closed,
   // the Valve is CloseING.
   // If the Valve is commanded to Close and the feedback shows it has Closed,
   // the Valve is Closed.
   67: [XIO(Mode.Sts_Hand) ,XIC(Cfg_UseOpenLS) ,XIC(Cfg_UseClosedLS) ][XIO(Wrk_Stop) [XIC(Wrk_Open) [XIO(Wrk_OpenFdbk) XIC(Wrk_ClosedFdbk) OTE(Sts_CmdToOpen) ,XIC(Wrk_TravelFdbk) OTE(Sts_Opening) ,XIC(Wrk_OpenFdbk) XIO(Wrk_ClosedFdbk) OTE(Sts_Opened) ] ,XIC(Wrk_Close) [XIO(Wrk_ClosedFdbk) XIC(Wrk_OpenFdbk) OTE(Sts_CmdToClose) ,XIC(Wrk_TravelFdbk) OTE(Sts_Closing) ,XIC(Wrk_ClosedFdbk) XIO(Wrk_OpenFdbk) OTE(Sts_Closed) ] ] ,XIC(Wrk_Stop) [OTE(Sts_Stopped) ,[XIC(Wrk_OpenFdbk) XIO(Wrk_ClosedFdbk) OTL(Wrk_Open) ,XIC(Wrk_ClosedFdbk) XIO(Wrk_OpenFdbk) OTL(Wrk_Close) ] OTU(Wrk_Stop) ] ];
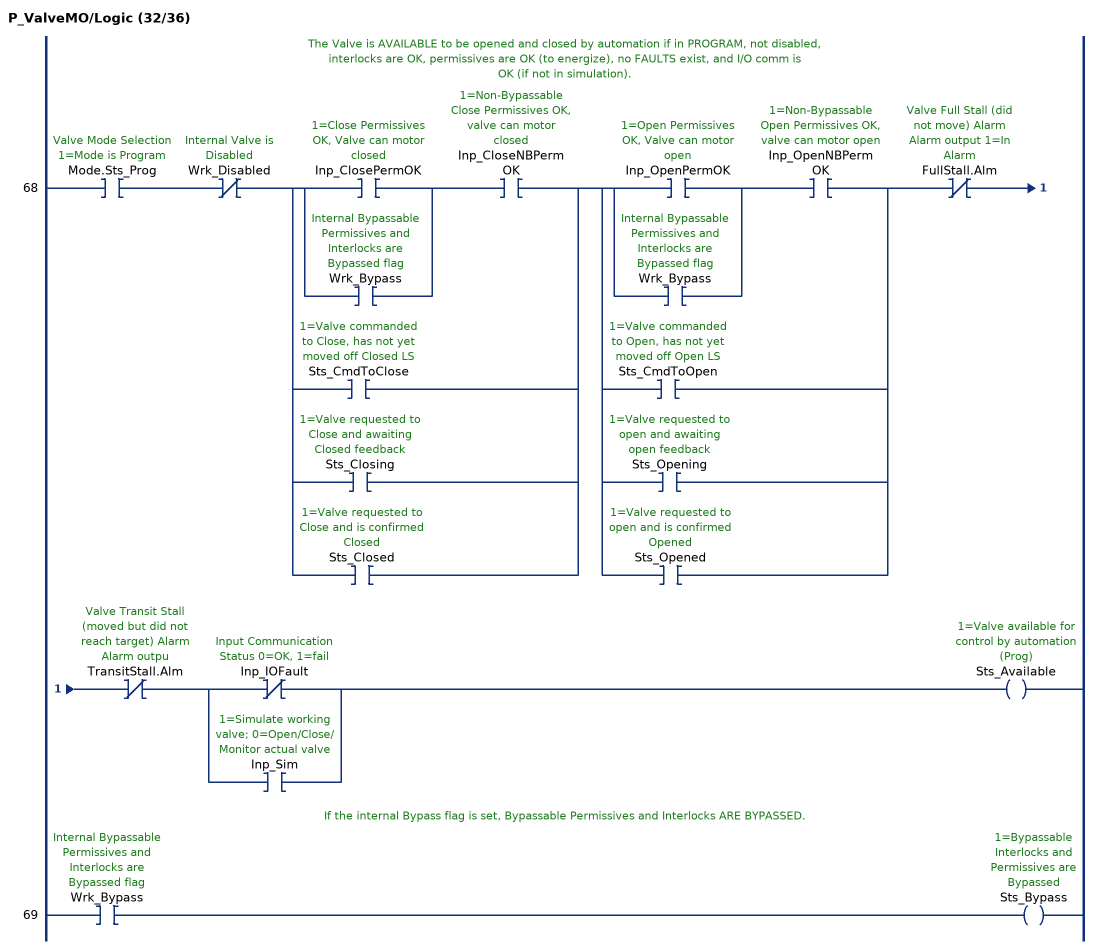
   // The Valve is AVAILABLE to be opened and closed by automation if in PROGRAM, not disabled,
   // interlocks are OK, permissives are OK (to energize), no FAULTS exist, and I/O comm is
   // OK (if not in simulation).
   68: XIC(Mode.Sts_Prog)XIO(Wrk_Disabled)[[XIC(Inp_ClosePermOK) ,XIC(Wrk_Bypass) ] XIC(Inp_CloseNBPermOK) ,XIC(Sts_CmdToClose) ,XIC(Sts_Closing) ,XIC(Sts_Closed) ][[XIC(Inp_OpenPermOK) ,XIC(Wrk_Bypass) ] XIC(Inp_OpenNBPermOK) ,XIC(Sts_CmdToOpen) ,XIC(Sts_Opening) ,XIC(Sts_Opened) ]XIO(FullStall.Alm)XIO(TransitStall.Alm)[XIO(Inp_IOFault) ,XIC(Inp_Sim) ]OTE(Sts_Available);
   // If the internal Bypass flag is set, Bypassable Permissives and Interlocks ARE BYPASSED.
   69: XIC(Wrk_Bypass)OTE(Sts_Bypass);
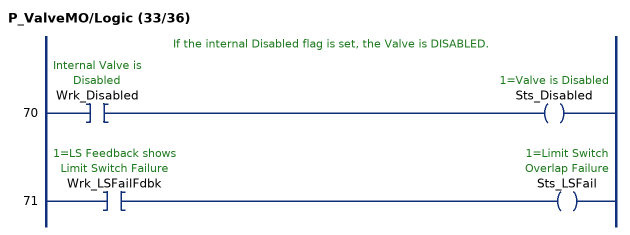
   // If the internal Disabled flag is set, the Valve is DISABLED.
   70: XIC(Wrk_Disabled)OTE(Sts_Disabled);
   71: XIC(Wrk_LSFailFdbk)OTE(Sts_LSFail);
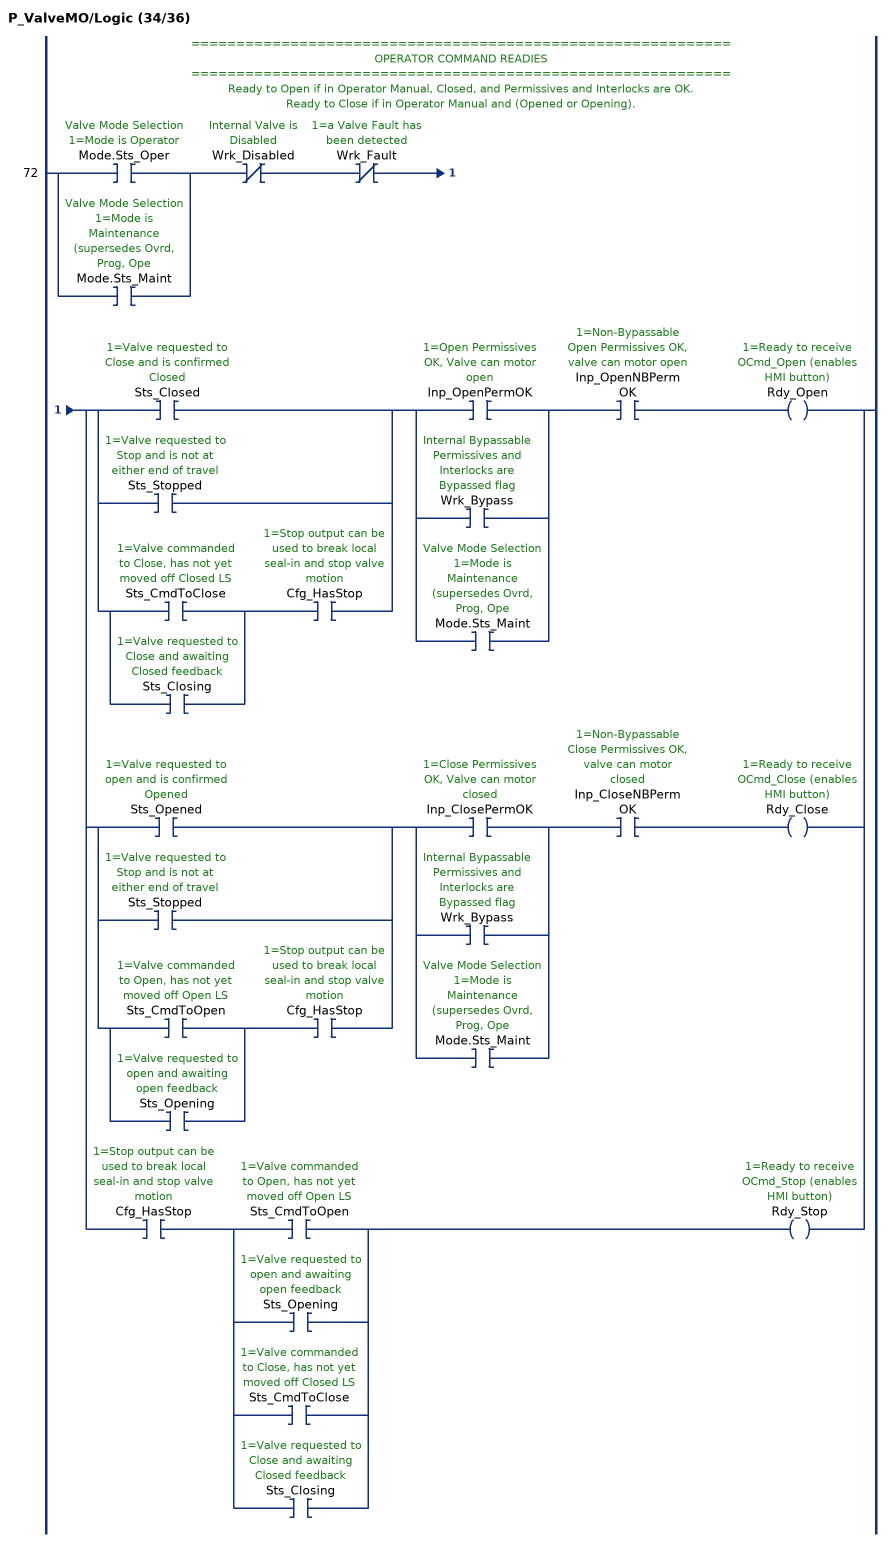
   // ============================================================
   // OPERATOR COMMAND READIES
   // ============================================================
   // Ready to Open if in Operator Manual, Closed, and Permissives and Interlocks are OK.
   // Ready to Close if in Operator Manual and (Opened or Opening).
   72: [XIC(Mode.Sts_Oper) ,XIC(Mode.Sts_Maint) ]XIO(Wrk_Disabled)XIO(Wrk_Fault)[[XIC(Sts_Closed) ,XIC(Sts_Stopped) ,[XIC(Sts_CmdToClose) ,XIC(Sts_Closing) ] XIC(Cfg_HasStop) ] [[XIC(Inp_OpenPermOK) ,XIC(Wrk_Bypass) ] ,XIC(Mode.Sts_Maint) ] XIC(Inp_OpenNBPermOK) OTE(Rdy_Open) ,[XIC(Sts_Opened) ,XIC(Sts_Stopped) ,[XIC(Sts_CmdToOpen) ,XIC(Sts_Opening) ] XIC(Cfg_HasStop) ] [[XIC(Inp_ClosePermOK) ,XIC(Wrk_Bypass) ] ,XIC(Mode.Sts_Maint) ] XIC(Inp_CloseNBPermOK) OTE(Rdy_Close) ,XIC(Cfg_HasStop) [XIC(Sts_CmdToOpen) ,XIC(Sts_Opening) ,XIC(Sts_CmdToClose) ,XIC(Sts_Closing) ] OTE(Rdy_Stop) ];
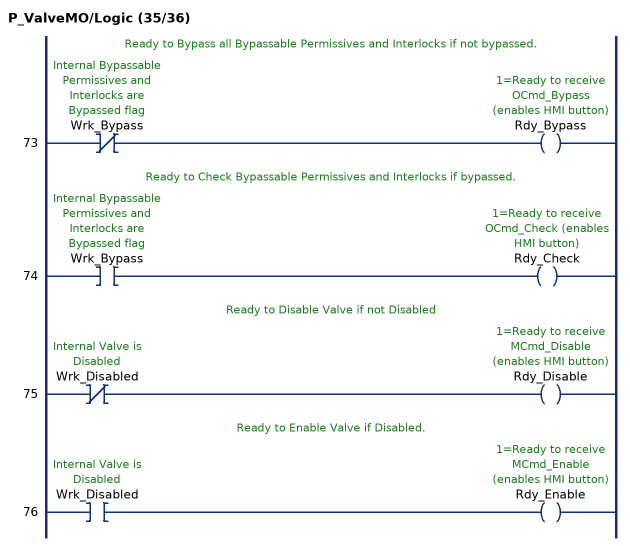
   // Ready to Bypass all Bypassable Permissives and Interlocks if not bypassed.
   73: XIO(Wrk_Bypass)OTE(Rdy_Bypass);
   // Ready to Check Bypassable Permissives and Interlocks if bypassed.
   74: XIC(Wrk_Bypass)OTE(Rdy_Check);
   // Ready to Disable Valve if not Disabled
   75: XIO(Wrk_Disabled)OTE(Rdy_Disable);
   // Ready to Enable Valve if Disabled.
   76: XIC(Wrk_Disabled)OTE(Rdy_Enable);
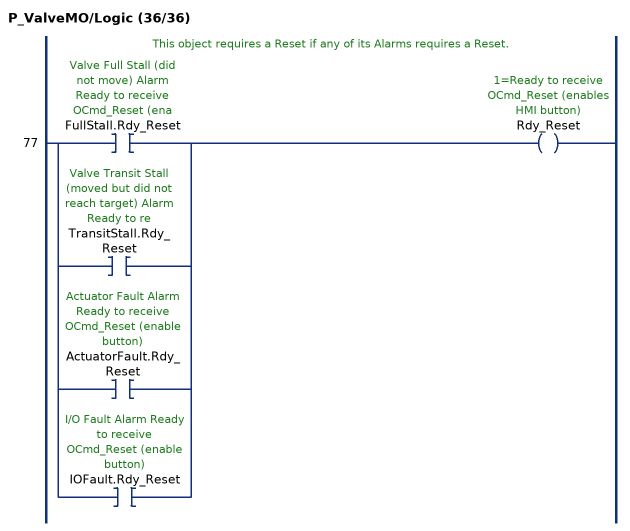
   // This object requires a Reset if any of its Alarms requires a Reset.
   77: [XIC(FullStall.Rdy_Reset) ,XIC(TransitStall.Rdy_Reset) ,XIC(ActuatorFault.Rdy_Reset) ,XIC(IOFault.Rdy_Reset) ]OTE(Rdy_Reset);
END_ROUTINE
